RoboDK station: Test preparion_syringe.rdk

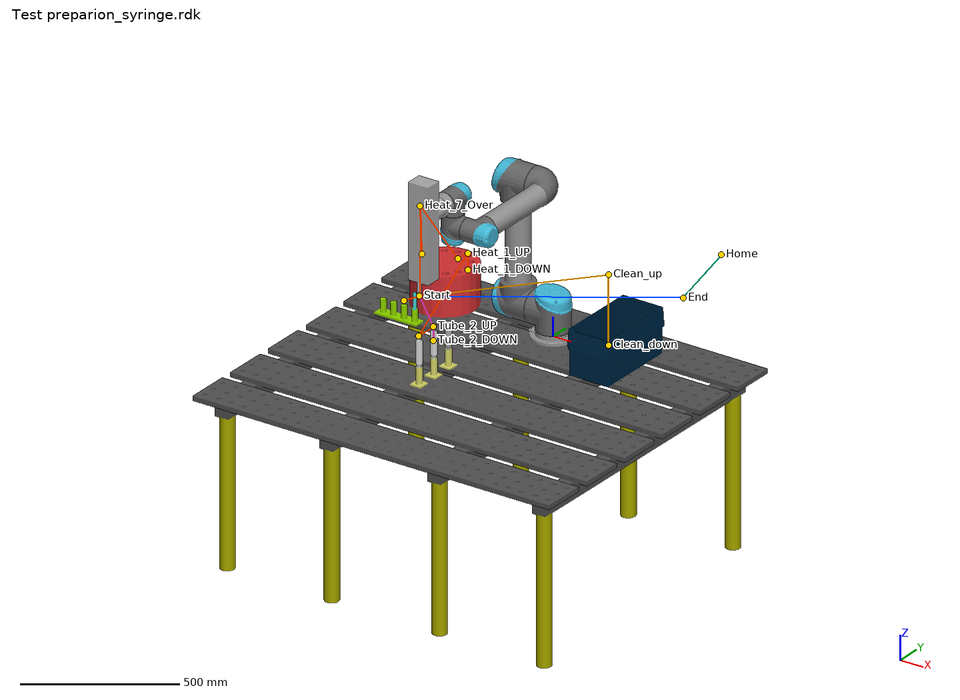
[picture v0: the station drawn from its stored meshes, robots at their saved joint values, targets as dots, program paths as lines]
Station Test preparion_syringe (saved by RoboDK 5.3.4). Poses are relative to the parent item; angles as X-Y-Z fixed-axis rotations.
  - frame UR5 Base at (-300, 0, 0) mm
    - robot UR5: 6 axes, payload 5 kg, reach 850 mm, repeatability 0.1 mm, weight 18.4 kg
        modified DH rows (alpha deg, a mm, theta deg, d mm): 0, 0, 0, 89.2; 90, 0, 180, 0; 0, 425, 0, 0; 0, 392.43, 0, 109; -90, 0, 0, 93.65; 90, 0, 180, 82
        joint limits [-360, -360, -360, -360, -360, -360] to [360, 360, 360, 360, 360, 360]; home [0, -90, -90, 0, 90, 0]; saved at [-90, -90, -90, 0, 90, -45]
      - tool Needle, TCP at (-189.46, 190.58, 100.42) mm, rotated rx 0 ry 0 rz 45 deg, size 76 x 107 x 390 mm, geometry from Needle.stp
  - frame World at (-300, 0, 0) mm
    - object Table_1 at (0, 0, 0) mm, size 1193.8 x 965.2 x 609.6 mm, geometry from welding_table.sld
    - object Table_2 at (0, 0, 0) mm, size 1193.8 x 965.2 x 609.6 mm, geometry from welding_table.sld
    - object Heater at (0, 0, 0) mm, size 225 x 140 x 222.7 mm, geometry from Heater.stl
    - object Fixture_2 at (0, 0, 0) mm, size 40 x 63 x 40 mm, geometry from Fixture_1.stl
    - object Test-tube-2 at (0, 0, 0) mm, size 22 x 147.5 x 22 mm, geometry from Test-tube.stl
    - object Test-tube-1 at (0, 0, 0) mm, size 22 x 147.5 x 22 mm, geometry from Test-tube.stl
    - object Fixture_1 at (0, 0, 0) mm, size 40 x 63 x 40 mm, geometry from Fixture_1.stl
    - object Test-tube-3 at (0, 0, 0) mm, size 22 x 147.5 x 22 mm, geometry from Test-tube.stl
    - object Fixture_3 at (0, 0, 0) mm, size 40 x 63 x 40 mm, geometry from Fixture_1.stl
    - object SFixture_2 at (0, 0, 0) mm, size 160 x 40 x 50 mm, geometry from Fixture_2.stp
    - object Smalltube at (0, 0, 0) mm, size 12 x 12 x 100 mm, geometry from Smalltube.stp
    - object Waterbox at (0, 0, 0) mm, size 166 x 315.8 x 161.6 mm, geometry from Box-400mmx200mm-Opened.sld
  - frame Calibration Target at (-300, 0, 0) mm
    - target Home (Cartesian target) at (587.71, 80.46, 417.27) mm, rotated rx -90 ry 45 rz -90 deg; joints [0, -91.734, -88.238, -0.028, 90, 0] of UR5
    - target End (Cartesian target) at (574.85, -109.79, 339.12) mm, rotated rx -90 ry 0 rz -90 deg; joints [0, -90, -90, 0, 90, -45] of UR5
    - target Start (Cartesian target) at (-109.79, -574.85, 339.12) mm, rotated rx -90 ry 0 rz -180 deg; joints [-90, -90, -90, 0, 90, -45] of UR5
  - frame Working at (-300, 0, 0) mm
    - target Tube_2_UP (Cartesian target) at (-146.27, -444.83, 170.09) mm, rotated rx -90 ry 0 rz 180 deg; joints [-97.702, -79.428, -124.924, 24.351, 97.702, -45] of UR5
    - target Tube_2_DOWN (Cartesian target) at (-146.27, -444.83, 121.16) mm, rotated rx -90 ry 0 rz 180 deg; joints [-97.702, -83.427, -129.822, 33.249, 97.702, -45] of UR5
    - target Tube_3_UP (Cartesian target) at (-146.27, -525.2, 170.09) mm, rotated rx -90 ry 0 rz 180 deg; joints [-95.976, -90.256, -115.256, 25.512, 95.976, -45] of UR5
    - target Heat_1_UP (Cartesian target) at (-339.42, 17.92, 187.09) mm, rotated rx -90 ry 0 rz 87.39 deg; joints [-139.411, -49.592, -137.823, 7.416, 46.8, -45] of UR5
    - target Heat_1_DOWN (Cartesian target) at (-339.42, 17.92, 129.53) mm, rotated rx -90 ry 0 rz 87.39 deg; joints [-139.411, -52.345, -145.624, 17.97, 46.8, -45] of UR5
    - target Heat_7_Over (Cartesian target) at (-507.32, -2.91, 314.25) mm, rotated rx -90 ry 0 rz 87.38 deg; joints [-158.304, -78.388, -103.974, 2.362, 65.68, -45] of UR5
    - target Smalltube (Cartesian target) at (-452.16, -169.78, 66.62) mm, rotated rx -90 ry 0 rz 87.36 deg; joints [-126.795, -92.977, -130.885, 43.862, 34.156, -45] of UR5
    - target Heat_7_DOWN (Cartesian target) at (-501.11, -3.19, 148.24) mm, rotated rx -90 ry 0 rz 87.38 deg; joints [-157.818, -84.032, -124.688, 28.721, 65.199, -45] of UR5
    - target Heat_2_UP (Cartesian target) at (-345.21, -27.46, 186.55) mm, rotated rx -90 ry 0 rz 87.37 deg; joints [-126.614, -52.17, -137.106, 9.275, 33.979, -45] of UR5
    - target Clean_up (Cartesian target) at (289.04, -109.79, 339.12) mm, rotated rx -90 ry 0 rz -90 deg; joints [0, -50.027, -115.315, -14.658, 90, -45] of UR5
    - target Clean_down (Cartesian target) at (289.04, -109.79, 92.8) mm, rotated rx -90 ry 0 rz -90 deg; joints [0, -54.112, -150.854, 24.966, 90, -45] of UR5
  - program Calibration (8 instructions, listed below)
  - program Position_Calibration (15 instructions, listed below)
  - program Move to Start point (4 instructions, listed below)
  - program Back to home (5 instructions, listed below)
  - program Draw from tube_2 (14 instructions, listed below)
  - program Cleaning the syringe (21 instructions, listed below)
  - program MainProgram (3 instructions, listed below)
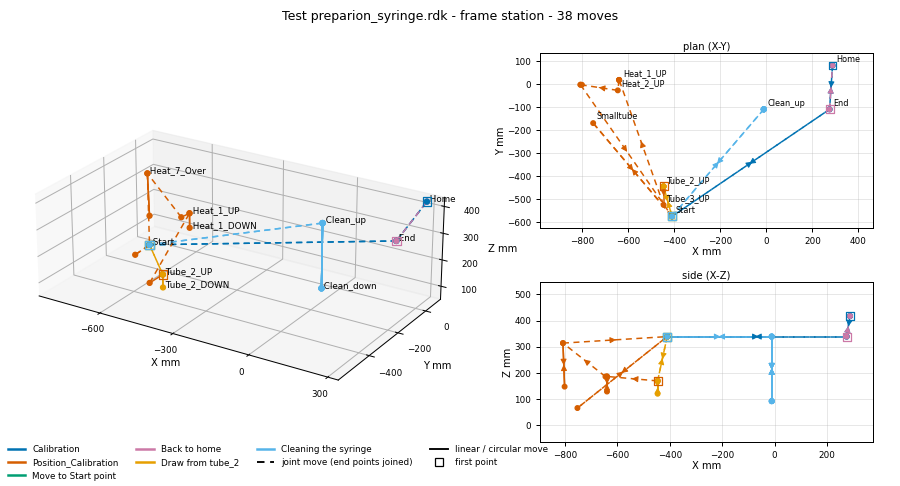
[picture p0: tool path of Test preparion_syringe.rdk in frame station, 38 of 38 moves have a stored position in this frame; points joined in program order, loops and branches not executed]

--- program Calibration (robot UR5) ---
  替换物体
  设置参考: Calibration Target
  设置工具: Needle
  MoveJ (Home)
  MoveJ (End)
  MoveJ (Start)
  MoveJ (End)
  MoveJ (Home)

--- program Position_Calibration (robot UR5) ---
  替换物体
  设置参考: Test -> Working
  设置工具: Needle
  MoveL (Tube_2_UP)
  MoveL (Tube_3_UP)
  MoveJ (Target 4) -> target Heat_1_UP
  MoveL (Target 5) -> target Heat_1_DOWN
  MoveL (Target 4) -> target Heat_1_UP
  MoveJ (Heat_2_UP)
  MoveJ (Target 9) -> target Heat_7_Over
  MoveL (Heat_7_DOWN)
  MoveL (Target 9) -> target Heat_7_Over
  MoveJ (Start)
  MoveJ (Target 9) -> target Smalltube
  MoveJ (Start)

--- program Move to Start point (robot UR5) ---
  替换物体
  设置参考: Calibration Target
  设置工具: Needle
  MoveJ (Start)

--- program Back to home (robot UR5) ---
  替换物体
  设置参考: Calibration Target
  设置工具: Needle
  MoveJ (End)
  MoveJ (Home)

--- program Draw from tube_2 (robot UR5) ---
  替换物体
  设置参考: Calibration Target
  设置工具: Needle
  Set speed (500.0 mm/s)
  MoveJ (Start)
  MoveJ (Tube_2_UP)
  暂停 500 ms
  Set speed (50.0 mm/s)
  MoveL (Tube_2_DOWN)
  Pause 2.5 s
  Set speed (50.0 mm/s)
  MoveL (Tube_2_UP)
  Set speed (500.0 mm/s)
  MoveJ (Start)

--- program Cleaning the syringe (robot UR5) ---
  替换物体
  设置参考: Calibration Target
  设置工具: Needle
  MoveJ (Start)
  MoveJ (Clean_up)
  MoveL (Clean_down)
  暂停 500 ms
  MoveL (Clean_up)
  MoveL (Clean_down)
  暂停 500 ms
  MoveL (Clean_up)
  MoveL (Clean_down)
  暂停 500 ms
  MoveL (Clean_up)
  MoveL (Clean_down)
  暂停 500 ms
  MoveL (Clean_up)
  MoveL (Clean_down)
  暂停 500 ms
  MoveL (Clean_up)
  MoveJ (Start)

--- program MainProgram (robot UR5) ---
  Call Move to Start point
  Call Draw from tube_2
  Call Move to Start point
